# EPICS substitutions: rga-01/asyn.substitutions
file /usr/lib/epics/db/asynRecord.db
{
	pattern { P     , R              , PORT      , ADDR , IMAX , OMAX }
	{ XF:23ID1-CT , "{Mir:3-RGAC:1}Asyn" , tsrv1-P7  , 0    , 80   , 80 }
	{ XF:23ID1-CT , "{Dif-RGAC:1}Asyn" , tsrv2-P7  , 0    , 80   , 80 }
}
